FUNCTION_BLOCK ActivateTrackTask IMPLEMENTS I_Task, I_Cyclic, I_Object, I_Abortable
VAR
	mcActivateTrack : Tc3_McCollisionAvoidance.MC_ActivateTrack;
	_Axis : REFERENCE TO Tc2_MC2.AXIS_REF;
	_newTrackId : OTCID;
	_Done : BOOL;
	_Error : BOOL;
	_ErrorId : UDINT;
END_VAR

{analysis -2}

METHOD Abort : HRESULT
mcActivateTrack.Execute := FALSE;
END_METHOD

PROPERTY AxisRef : reference to Axis_ref
GET
AxisRef	REF= _Axis;
END_GET
SET
_Axis REF= AxisRef;
END_SET
END_PROPERTY

PROPERTY Busy : BOOL
GET
Busy := mcActivateTrack.Busy;
END_GET
END_PROPERTY

METHOD Cycle : HRESULT
VAR_INPUT
END_VAR
IF NOT __ISVALIDREF(_Axis) THEN
	Cycle := -1;
	RETURN;
END_IF
_Done := mcActivateTrack.Done OR _Done;
_Error := mcActivateTrack.Error OR _Error;
IF mcActivateTrack.ErrorId <> 0 THEN
	_ErrorId := mcActivateTrack.ErrorId;
END_IF
_newTrackId := mcActivateTrack.TrackId;
mcActivateTrack(Axis := _Axis);
mcActivateTrack.Execute := FALSE;
END_METHOD

PROPERTY Done : BOOL
GET
Done := _Done;
END_GET
END_PROPERTY

PROPERTY Error : BOOL
GET
Error := _Error;
END_GET
END_PROPERTY

METHOD PUBLIC Execute : HRESULT
VAR_INPUT
	Track : I_XtsTrack;
END_VAR
IF mcActivateTrack.Execute THEN
	Execute := -1;
	RETURN;
END_IF

IF Track = 0 THEN
	Execute := -2;
	RETURN;
END_IF

IF NOT __ISVALIDREF(_Axis) THEN
	Execute := - 3;
	RETURN;
END_IF;

IF _Axis.Status.Disabled THEN
	Execute := -4;
	RETURN;
END_IF

IF _Axis.NcToPlc.SetVelo <> 0.0 THEN
	Execute := -5;
	RETURN;
END_IF

mcActivateTrack.Execute := TRUE;
mcActivateTrack.TrackId := Track.MyOTCID;
_Error := FALSE;
_ErrorId := 0;
_Done := FALSE;
END_METHOD

PROPERTY PUBLIC NewTrackId : OTCID
GET
NewTrackId := _newTrackId;
END_GET
END_PROPERTY

METHOD RegisterWithParent
VAR_INPUT
	Parent	: Base_Library.I_HostObjects;
END_VAR
Parent.RegisterCyclic(THIS^);
Parent.RegisterAbortable(THIS^);
Parent.RegisterTask(THIS^);
END_METHOD

END_FUNCTION_BLOCK

(* stored: Version 1.1.0.1
   POU ActivateTrackTask: Id {03f53080-a7f0-4bc3-a76f-2f27947df261}, SpecialFunc None
   Method Abort: Id {12b22699-a9ca-4822-aec7-46d8d5f2084b}
   Property AxisRef: Id {cd922916-f6a4-41a1-9317-bcc0a2f58821}
   Get Get: Id {f8bd9ae9-fd4a-4869-b258-23c1451a49b1}
   Set Set: Id {2d897f7c-ffe5-43a2-ab4e-fd6eede8b200}
   Property Busy: Id {23074907-2ae6-43d6-952f-8555fe23ba80}
   Get Get: Id {4a3a6bc3-a08b-4d30-bf35-0fdb74a6daa4}
   Method Cycle: Id {57b0f6ac-3d25-41af-b69c-d2ca0682dcf2}
   Property Done: Id {c8440faf-d9f2-4d0f-8b0f-12623384efd8}
   Get Get: Id {567704db-7419-4756-aae9-b62178c2fc84}
   Property Error: Id {cd1cdc81-f00a-4514-9adc-1c583f307c6e}
   Get Get: Id {a7583719-1e76-4918-b599-0ba47213ed74}
   Method Execute: Id {b92caa48-be0c-4823-bb15-e823e8bc1934}
   Property NewTrackId: Id {84df412b-7c3c-4f84-98eb-ff5f562dbb1a}
   Get Get: Id {cb5898cd-640b-468a-893b-247f32481adb}
   Method RegisterWithParent: Id {492c1dba-ce80-4d69-a740-59e5f54b10be} *)
